// TIA Portal V20 export
TYPE "typeCmControlNode"
// stored: Namespace Unit1.Em7
   STRUCT
      Interlock { ExternalWritable := 'False'} : "Unit1.Em7.typeCmControlNodeInterlock";
      brakeTest { ExternalWritable := 'False'} : "Unit1.Em7.typeCmControlNodeBrakeTest";
   END_STRUCT;
END_TYPE
